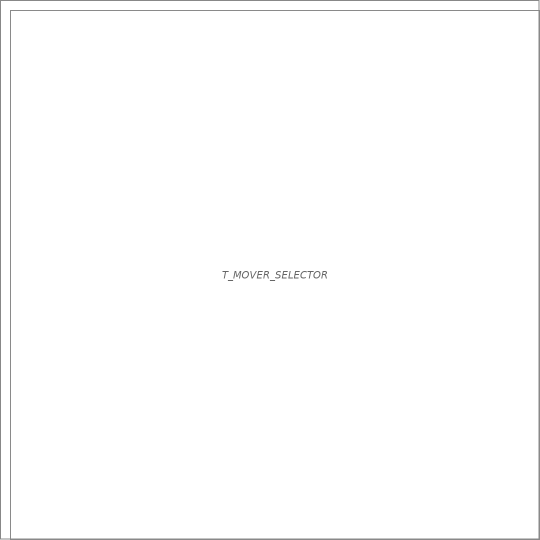
VISUALIZATION SELECTOR_VISU  // 540x540
    Frame (10,10 530x530)
        shows T_MOVER_SELECTOR(Control := GVL_XTS.MoverSelectorCtrl, State := GVL_XTS.MoverSelectorState, sState := VISU_XTS.sSelectorState, sResult := VISU_XTS.sSelectorResult)
END_VISUALIZATION

(* stored: Version 1.1.0.1, ProductVersion 3.1.4026.20
   Visu SELECTOR_VISU: Id {e9505c66-7e20-437e-9859-be1cb953ae7b} *)
